INTERFACE ISensor

PROPERTY Value : LREAL
GET
END_GET
END_PROPERTY

END_INTERFACE

(* stored: Version 1.1.0.1
   Itf ISensor: Id {779a4d97-b574-0547-2303-8c3847733ce4}
   Property Value: Id {f836dc53-abda-030b-3dde-0f79dabdd6d6}
   Get Get: Id {2ba26cfc-c861-03af-0f77-26ce8a2e7fec} *)
